ADAPTER ASR2 (* bidirectional Adapter Interface for 2 Events *)
  (* Standard: 61499-1; Description: Copyright (c) 2025 HR Agrartechnik GmbH This program and the accompanying materials are made available under the terms of the Eclipse Public License 2.0 which is available at https://www.eclipse.org/legal/epl-2.0/ SPDX-License-Identifier: EPL-2.0 *)
  (* Version 1.0, 2025-05-27, Franz Höpfinger, HR Agrartechnik GmbH *)
  PACKAGE adapter::types::bidirectional;
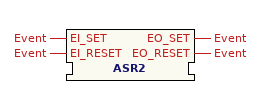
  EVENT_INPUT
    EI_SET; (* Set / Switch on *)
    EI_RESET; (* Reset / Switch off *)
  END_EVENT
  EVENT_OUTPUT
    EO_SET; (* Set / Switch on *)
    EO_RESET; (* Reset / Switch off *)
  END_EVENT
END_ADAPTER
